// TIA Portal V18 export
TYPE "MEStoPLC_AlarmMassage_ext"
// stored: IsFailsafeCompliant false
   STRUCT
      ErrorCode : Int;   // Process error code
      StatusBits : DInt;   // The StatusBits set by the PLC and by the ACC rework PC
      Cycle_ID : DInt;   // Spare
      Unit_ParttypeID : Int;   // Spare
      "Transfer time" : String[60];   // 工位1执行时间日期
   END_STRUCT;
END_TYPE
